Staubli VAL3: tool.pjx

--- tool.pjx ---
Parameters version=s7.2.1 stackSize=5000 millimeterUnit=true
Program file=checkPoint.pgx
Program file=compose.pgx
Program file=delete.pgx
Program file=getAction.pgx
Program file=getName.pgx
Program file=getSize.pgx
Program file=getTool.pgx
Program file=goToPoint.pgx
Program file=here.pgx
Program file=new.pgx
Program file=save.pgx
Program file=setAction.pgx
Program file=setName.pgx
Program file=setTool.pgx
Data file=tool.dtx
Library alias=io path=Disk://io/io.pjx
Library alias=saveTool path=Disk://saveTool/saveTool.pjx
Library alias=use path=Disk://kernel/userPage/userPage.pjx

--- tool.dtx ---
string pathGun
pointRx pPoint = {wrist=wfree, fatherId=world[0]}

--- checkPoint.pgx ---
public program checkPoint(bool& x_bCheck[])
begin
  x_bCheck=saveTool:bCheck
end

--- compose.pgx ---
public program compose(num x_nIndexGun)
  local trsf tPar
  local tool tGun
  local point pPoint
begin
  pPoint=here(flange,world)
  tPar=!pPoint.trsf*saveTool:rif2.trsf
  tGun.trsf=tPar
  call setTool(tGun,x_nIndexGun)
end

--- delete.pgx ---
public program delete(num x_nIndexGun)
begin
  $ddel(saveTool:gun,x_nIndexGun)
  $ddel(saveTool:name,x_nIndexGun)
  $ddel(saveTool:sActionOFF,x_nIndexGun)
  $ddel(saveTool:sActionON,x_nIndexGun)
end

--- getAction.pgx ---
public program getAction(string& x_sInstruction[], bool x_bType, num x_nIndex)
  local string l_sInstruction
begin
  // get the instruction and fill as an array
  if x_nIndex>=0
    if x_bType
      // take gun ON
      l_sInstruction=saveTool:sActionON[x_nIndex]
    else
      // take gun OFF
      l_sInstruction=saveTool:sActionOFF[x_nIndex]
    endIf
    // make it to three element
    if l_sInstruction==""
      l_sInstruction=",,"
    endIf
    call use:stringToArray(l_sInstruction,x_sInstruction)
  endIf
end

--- getName.pgx ---
public program getName(string& x_sName[], num x_nIndex)
begin
  x_sName=saveTool:name[x_nIndex]
end

--- getSize.pgx ---
public program getSize(num& nSize[])
begin
  nSize=size(saveTool:gun)
end

--- getTool.pgx ---
public program getTool(tool& x_tTool[], num x_nIndex)
begin
  //
  x_tTool=saveTool:gun[x_nIndex]
end

--- goToPoint.pgx ---
public program goToPoint(num x_nIndexGun)
begin
  resetMotion()
  if x_nIndexGun==0
    movej(saveTool:rif2,saveTool:gun[x_nIndexGun],{25,25,25,9999,9999,off,50,50})
  else
    pPoint.trsf=position(saveTool:rif2,world)
    pPoint.config={sfree,efree,wfree}
    movej(pPoint,saveTool:gun[x_nIndexGun],{25,25,25,9999,9999,off,50,50})
  endIf
end

--- here.pgx ---
public program here()
begin
  saveTool:rif2=here(saveTool:gun[0],world)
  saveTool:bCheck=true
end

--- new.pgx ---
public program new(trsf& tPar[])
  local num nSize
  local tool tGun
begin
  // only fifo polit
  call getSize(nSize)
  // TRSF
  $dins(saveTool:gun,nSize)
  tGun.trsf=tPar
  call setTool(tGun,nSize)
  // NAME
  $dins(saveTool:name,nSize)
  call setName("",nSize)
  // ACTION
  $dins(saveTool:sActionON,nSize)
  $dins(saveTool:sActionOFF,nSize)
end

--- save.pgx ---
public program save(num& x_nResult[])
  local num i
begin
  x_nResult=saveTool:libSave()
  if x_nResult!=0
    delay(0.5)
    x_nResult=saveTool:libSave()
  endIf
end

--- setAction.pgx ---
public program setAction(string& x_sAction[], num x_nIndex, bool x_bType)
  local string l_sInstruction
  local num i
begin
  // get the instruction and fill as an array
  if x_nIndex>=0
    if x_sAction[0]!="" or x_sAction[1]!="" or x_sAction[2]!=""
      // array to string
      l_sInstruction=x_sAction[0]
      for i=1 to size(x_sAction)-1
        l_sInstruction=l_sInstruction+"^"+x_sAction[i]
      endFor
    else
      // set empty
      l_sInstruction=""
    endIf
    // save the data
    if x_bType
      // take gun ON
      saveTool:sActionON[x_nIndex]=l_sInstruction
    else
      // take gun OFF
      saveTool:sActionOFF[x_nIndex]=l_sInstruction
    endIf
  endIf
end

--- setName.pgx ---
public program setName(string x_sName, num x_nIndex)
begin
  saveTool:name[x_nIndex]=x_sName
end

--- setTool.pgx ---
public program setTool(tool tParGun, num x_nIndex)
begin
  saveTool:gun[x_nIndex].trsf=tParGun.trsf
end
